// TIA Portal V18 program export: 1 tag tables, 0 data types, 2 data blocks, 3 code blocks (in call order from the OBs), 2 instance data blocks

VAR_GLOBAL   // PLC tag table "Default tag table"
   System_Byte AT %MB1 : Byte;
   FirstScan AT %M1.0 : Bool;
   DiagStatusUpdate AT %M1.1 : Bool;
   AlwaysTRUE AT %M1.2 : Bool;
   AlwaysFALSE AT %M1.3 : Bool;
   Clock_Byte AT %MB0 : Byte;
   Clock_10Hz AT %M0.0 : Bool;
   Clock_5Hz AT %M0.1 : Bool;
   "Clock_2.5Hz" AT %M0.2 : Bool;
   Clock_2Hz AT %M0.3 : Bool;
   "Clock_1.25Hz" AT %M0.4 : Bool;
   Clock_1Hz AT %M0.5 : Bool;
   "Clock_0.625Hz" AT %M0.6 : Bool;
   "Clock_0.5Hz" AT %M0.7 : Bool;
END_VAR

DATA_BLOCK "Dest_DB"   // DB4
{ S7_Optimized_Access := 'FALSE' }
   VAR
      IN1 : Array[0..5] of Int;
      IN2 : Int;
      IN3 : Int;
      IN4 : Int;
   END_VAR
BEGIN
END_DATA_BLOCK

DATA_BLOCK "Source_DB"   // DB1
{ S7_Optimized_Access := 'FALSE' }
   VAR
      IN1 : Array[0..5] of Int;
      IN2 : Int;
      IN3 : Int;
      IN4 : Int;
      OUT : Int;
   END_VAR
BEGIN
END_DATA_BLOCK

ORGANIZATION_BLOCK "Main"   // OB1, LAD, ProgramCycle
TITLE = "Main Program Sweep (Cycle)"
{ S7_Optimized_Access := 'TRUE' }
// stored: SetENOAutomatically false
   VAR_INPUT
      Initial_Call : Bool;   // Initial call of this OB
      Remanence : Bool;   // =True, if remanent data are available
   END_VAR
   VAR_TEMP   // added for the SCL form of the ladder/FBD networks
      _w1 : Bool;
   END_VAR
BEGIN

REGION Network 1
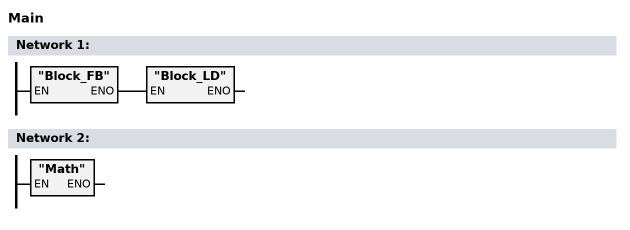
   RUNG wire#powerrail
      "Block_FB"()
      "Block_LD"()
   END_RUNG
   // the same network as SCL:
   "Block_FB"(ENO => #_w1);
   IF #_w1 THEN "Block_LD"(); END_IF;
END_REGION

REGION Network 2
   RUNG wire#powerrail
      "Math"()
   END_RUNG
   // the same network as SCL:
   "Math"();
END_REGION
END_ORGANIZATION_BLOCK

FUNCTION "Block_FB" : Void   // FC1, FBD
{ S7_Optimized_Access := 'TRUE' }
// stored: SetENOAutomatically false
   VAR_TEMP
      "A" : Bool;
      "B" : Bool;
      Q : Bool;
   END_VAR
BEGIN

REGION Network 1
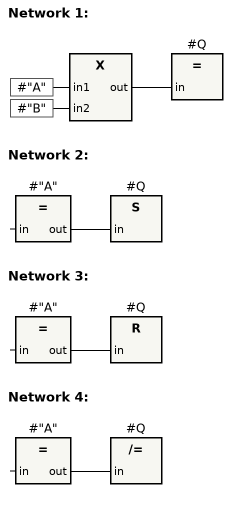
   #Q := #"A" XOR #"B";
END_REGION

REGION Network 2
   #"A" := TRUE;
   #Q := TRUE;
END_REGION

REGION Network 3
   #"A" := TRUE;
   #Q := FALSE;
END_REGION

REGION Network 4
   #"A" := TRUE;
   #Q := NOT TRUE;
END_REGION
END_FUNCTION

FUNCTION "Block_LD" : Void   // FC2, LAD
{ S7_Optimized_Access := 'TRUE' }
// stored: SetENOAutomatically false
   VAR_TEMP
      "A" : Bool;
      "B" : Bool;
      C : Bool;
      D : Bool;
      QU : Bool;
      QD : Bool;
      PT : Time;
      ET : Time;
      PV : Int;
      CV : Int;
   END_VAR
BEGIN

REGION Network 1
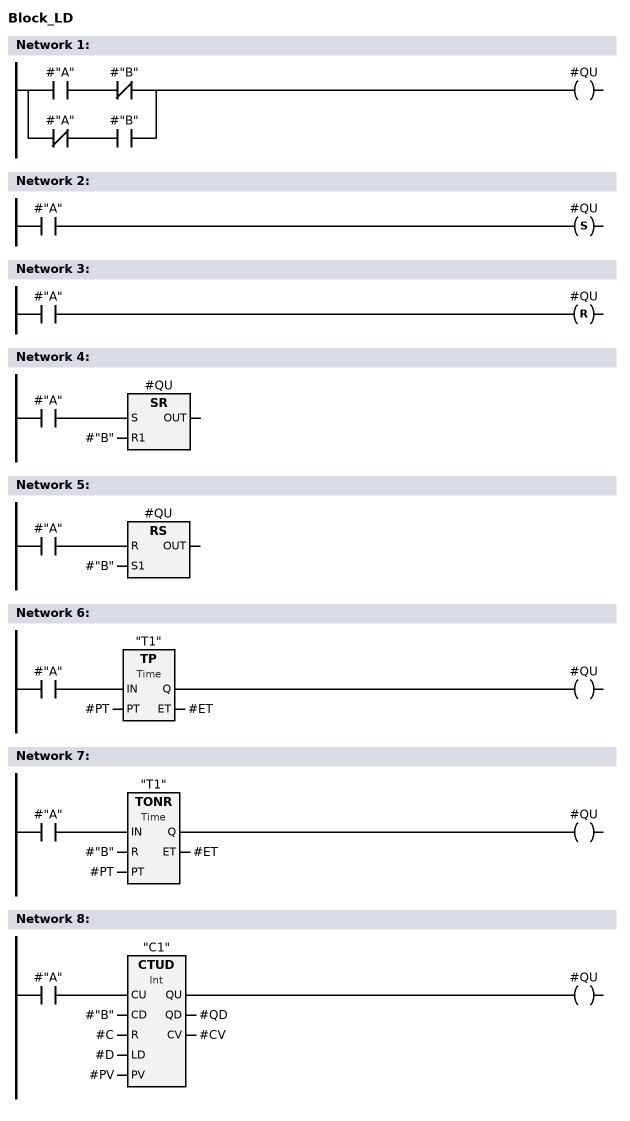
   RUNG wire#powerrail
      Contact( #"A" )
      I_Contact( #"B" )
      wire#w1
      Coil( #QU )
   END_RUNG
   RUNG wire#powerrail
      I_Contact( #"A" )
      Contact( #"B" )
   END_RUNG wire#w1
   // the same network as SCL:
   #QU := (#"A" AND NOT #"B") OR (NOT #"A" AND #"B");
END_REGION

REGION Network 2
   RUNG wire#powerrail
      Contact( #"A" )
      S_Coil( #QU )
   END_RUNG
   // the same network as SCL:
   IF #"A" THEN #QU := TRUE; END_IF;
END_REGION

REGION Network 3
   RUNG wire#powerrail
      Contact( #"A" )
      R_Coil( #QU )
   END_RUNG
   // the same network as SCL:
   IF #"A" THEN #QU := FALSE; END_IF;
END_REGION

REGION Network 4
   RUNG wire#powerrail
      Contact( #"A" )
      S_SR(operand := #QU, r1 := #"B")
   END_RUNG
   // the same network as SCL:
   IF #"A" THEN
       #QU := TRUE;   // SR flip-flop
   END_IF;
   IF #"B" THEN #QU := FALSE; END_IF;
END_REGION

REGION Network 5
   RUNG wire#powerrail
      Contact( #"A" )
      S_RS(operand := #QU, s1 := #"B")
   END_RUNG
   // the same network as SCL:
   IF #"A" THEN
       #QU := FALSE;   // RS flip-flop
   END_IF;
   IF #"B" THEN #QU := TRUE; END_IF;
END_REGION

REGION Network 6
   RUNG wire#powerrail
      Contact( #"A" )
      { S7_Templates := "time_type := Time" } "T1".TP(pt := #PT, et => #ET)
      Coil( #QU )
   END_RUNG
   // the same network as SCL:
   "T1".TP(IN := #"A", PT := #PT, ET => #ET);
   #QU := "T1".Q;
END_REGION

REGION Network 7
   RUNG wire#powerrail
      Contact( #"A" )
      { S7_Templates := "time_type := Time" } "T1".TONR(r := #"B", pt := #PT, et => #ET)
      Coil( #QU )
   END_RUNG
   // the same network as SCL:
   "T1".TONR(IN := #"A", R := #"B", PT := #PT, ET => #ET);
   #QU := "T1".Q;
END_REGION

REGION Network 8
   RUNG wire#powerrail
      Contact( #"A" )
      { S7_Templates := "value_type := Int" } "C1".CTUD(cd := #"B", r := #C, ld := #D, pv := #PV, qd => #QD, cv => #CV)
      Coil( #QU )
   END_RUNG
   // the same network as SCL:
   "C1".CTUD(CU := #"A", CD := #"B", R := #C, LD := #D, PV := #PV, QD => #QD, CV => #CV);
   #QU := "C1".QU;
END_REGION
END_FUNCTION

DATA_BLOCK "C1"   // DB3
{ S7_Optimized_Access := 'TRUE' }
// stored: InstanceOfName IEC_COUNTER, OfSystemLibElement IEC_COUNTER, OfSystemLibVersion 1.0
"IEC_COUNTER"
   // VAR RETAIN
   //    CU : Bool;
   //    CD : Bool;
   //    R : Bool;
   //    LD : Bool;
   //    QU : Bool;
   //    QD : Bool;
   //    PV : Int;
   //    CV : Int;
   // END_VAR
BEGIN
END_DATA_BLOCK

DATA_BLOCK "T1"   // DB2
{ S7_Optimized_Access := 'TRUE' }
// stored: InstanceOfName IEC_TIMER, OfSystemLibElement IEC_TIMER, OfSystemLibVersion 1.0
"IEC_TIMER"
   // VAR
   //    PT : Time;
   //    ET { ExternalWritable := 'False'} : Time;
   //    IN : Bool;
   //    Q { ExternalWritable := 'False'} : Bool;
   // END_VAR
BEGIN
END_DATA_BLOCK
